FUNCTION_BLOCK FB_Bel_Taster
VAR_INPUT
END_VAR
VAR_OUTPUT
	Betrieb			: BOOL:=TRUE;

END_VAR
VAR
	IN_Bin	AT %I* : BOOL;

	Taster			: R_TRIG;
	Halter			: RS;
	Licht_Schalten	: SINT := 2;

	Taster_Virtuell	: TP;
	Taste			: BOOL:=TRUE;

END_VAR
VAR // added by the converter: edge detectors and wires of the graphical bodies
    _w1, _w2, _w3 : ANY;
    _w4, _w5 : BOOL;
END_VAR

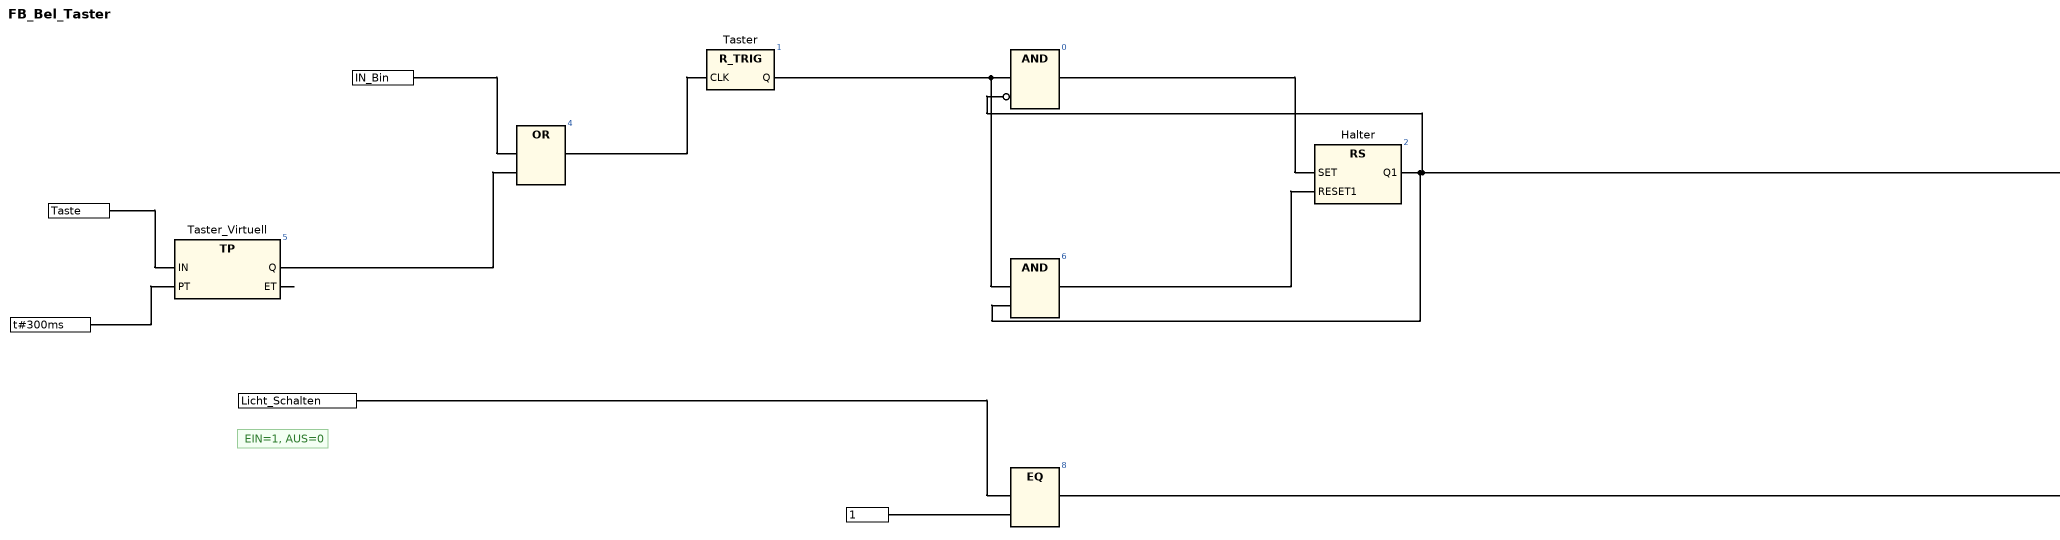
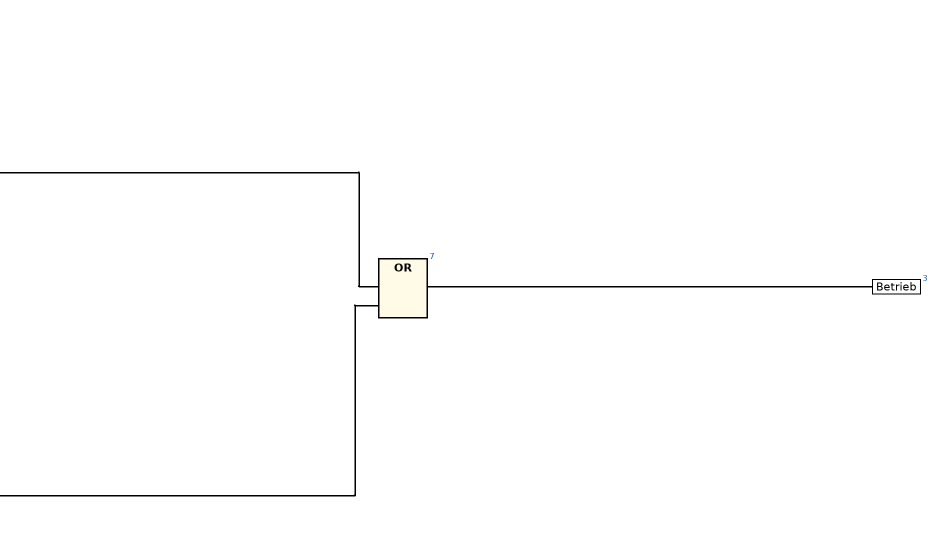
_w1 := Taster.Q AND NOT Halter.Q1;
Taster(CLK := _w2); // R_TRIG
Halter(SET := _w1, RESET1 := _w3); // RS
Betrieb := _w4;
_w2 := IN_Bin OR Taster_Virtuell.Q;
Taster_Virtuell(IN := Taste, PT := t#300ms); // TP
_w3 := Taster.Q AND Halter.Q1;
_w4 := Halter.Q1 OR _w5;
//  EIN=1, AUS=0
_w5 := Licht_Schalten = 1;

END_FUNCTION_BLOCK

(* stored: Version 1.1.0.1, ProductVersion 3.1.4024.9
   POU FB_Bel_Taster: Id {3d7e474e-f045-4242-9a14-0c29d4c9e5c2}, SpecialFunc None *)
